FUNCTION_BLOCK FB_IMPLICATION
VAR_INPUT
	Antecedent: REAL;
	X:REAL;
	FISOutputMf: MEMBERSHIP_FUNCTION;
END_VAR
VAR_OUTPUT
	RuleFuzzySet:REAL;
END_VAR

RuleFuzzySet :=fuzzyAND(Minimum,fMembershipDegree(x,FISOutputMf),Antecedent);

END_FUNCTION_BLOCK

(* stored: Version 1.1.0.1, ProductVersion 3.1.4024.6
   POU FB_IMPLICATION: Id {00c0c73f-264e-4bea-a4a3-7a9174640c0c}, SpecialFunc None *)
